{attribute 'qualified_only'}
{attribute 'strict'}
TYPE E_PickerFixedState :
(
	Idle        := 0,
	InPickedPos := 1,
	PartPicked 	:= 2,
	InPlacedPos := 3,
	PartPlaced  := 4
);
END_TYPE

(* stored: Version 1.1.0.1, ProductVersion 3.1.4024.12
   DUT E_PickerFixedState: Id {d35d3d88-f837-4e3a-8b00-81fecbb0a4b7} *)
